# B&R Automation Studio project OpcUaServer_Reading-SessionDiagnosticsArray
Automation Studio 4.9

## Configuration Config1

CPU PC_any, AutomationRuntime L4.93, Build 4.1.2, Vc V4.73.3

### Task classes (Cpu.sw)
```
Cyclic#1:
  Program <- Program.prg
  UASessDiag <- UASessDiag.prg
Binaries: udbdef, FWRules, TCData, sysconf, Role, User, iomap, ashwd, asfw, arconfig, ashwac
Libraries: AsOpcUac, runtime, standard, astime, asieccon
```

### Hardware
```
PC : PC_any v1.1.1.0 (OrderNumber=PC)
  ConfigurationID = uaserver_Config1
  FileDevice1
  FileDeviceName1 = USER
  FileDevicePath1 = USER_PATH
  ActivateOpcUa = 1
  OpcUaPort = 4841
  OpcUaInformationModels_PV_Version = 1
```

## Configuration Config2

CPU X20CP3585, AutomationRuntime J4.93, Build 4.1.2, Vc V4.73.3

### Task classes (Cpu.sw)
```
Cyclic#1:
  Program <- Program.prg
Cyclic#4:
  UASessDiag <- UASessDiag.prg
Libraries: AsIODiag, runtime
```

### Hardware
```
X20CP3585 : X20CP3585 v1.10.0.0
  Connector IF2:
    ActivateDevice = 1
    Mode = Manual
    InternetAddress = 10.24.153.43
    SubnetMask = 255.255.255.192
    ActivateIna = 0
    ActivateSnmp = 2
  ConfigurationID = uaserver_Config2
  FileDevice1
  FileDeviceName1 = USER
  FileDevicePath1 = USER_PATH
  EthernetDefaultGateway = 10.24.153.1
  ActivateOpcUa = 1
  OpcUaInformationModels_PV_Version = 1
```

## Logical view

Binary libraries used (declarations not repeated): operator, runtime, astime, AsIecCon, AsOpcUac, standard, AsIODiag


### Program Logical/Program (IEC)

#### Variables.var
```iecst
VAR
	i : DINT;
END_VAR
```

#### Main.st
```iecst
PROGRAM _INIT
	i := 0;

END_PROGRAM

PROGRAM _CYCLIC
	i := i + 1;

END_PROGRAM

PROGRAM _EXIT
	(* Insert code here *)

END_PROGRAM
```

### Program Logical/UASessDiag (IEC) - Read OPC UA session diagnostic

#### ReadSessionDiagnosticsArray.st - Cyclic code
```iecst
PROGRAM _INIT
	step := RSD_INIT;

	(* NodeId for Root/Objects/Server/ServerDiagnostics/SessionsDiagnosticsSummary/SessionDiagnosticsArray is i=3707. *)
	ServerDiagnosticNodeID.NamespaceIndex := 0;
	ServerDiagnosticNodeID.IdentifierType := UAIdentifierType_Numeric;
	ServerDiagnosticNodeID.Identifier := '3707';

	ServerDiagnosticVariable := 'SessionDiagnosticsArray';
	SessionDiagnosticsArray;
	tonRepeat.PT := T#5s;

	timeout := T#5s;
END_PROGRAM

PROGRAM _CYCLIC
	CASE step OF
		RSD_INIT:
		ErrorID := 0;
		IF DiagCpuIsSimulated() THEN
			fbUAConnect.ServerEndpointUrl := 'opc.tcp://localhost:4841';
		ELSE
			fbUAConnect.ServerEndpointUrl := 'opc.tcp://localhost:4840';
		END_IF
		fbUAConnect( Execute := FALSE,
				SessionConnectInfo := SessionConnectInfo,
				Timeout := timeout,
		); // reset fb
		fbUAConnect( Execute := TRUE );
		step := RSD_W_CONNECT;

		RSD_W_CONNECT:
		IF fbUAConnect.Done THEN (* ok *)
			fbUaNodeGetHandle( Execute := FALSE,
							ConnectionHdl := fbUAConnect.ConnectionHdl,
							NodeID := ServerDiagnosticNodeID,
							Timeout := timeout );
			fbUaNodeGetHandle( Execute := TRUE );
			fbUAConnect( Execute := FALSE ); (* reset fb *)
			step := RSD_W_NODE_HANDLE;
		ELSIF fbUAConnect.Error THEN (* error *)
			ErrorID := fbUAConnect.ErrorID;
			fbUAConnect( Execute := FALSE ); (* reset fb *)
			step := RSD_ERROR_CONNECT_TO_SERVER;
		ELSE (* busy *)
			fbUAConnect();
		END_IF

		RSD_W_NODE_HANDLE:
		IF fbUaNodeGetHandle.Done THEN (* ok *)
			fbUaRead( ConnectionHdl := fbUAConnect.ConnectionHdl,
					  NodeHdl := fbUaNodeGetHandle.NodeHdl,
					  Variable := ServerDiagnosticVariable,
					  Timeout := timeout
					);
			fbUaRead( Variable := ServerDiagnosticVariable, Execute := TRUE );
			fbUaNodeGetHandle( Execute := FALSE ); (* reset fb *)
			step := RSD_W_DIAGNOSTIC_READ;
		ELSIF fbUaNodeGetHandle.Error THEN (* error *)
			ErrorID := fbUaNodeGetHandle.Error;
			fbUaNodeGetHandle( Execute := FALSE ); (* reset fb *)
			step := RSD_ERROR_GET_NODE_HANDLE;
		ELSE (* busy *)
			fbUaNodeGetHandle();
		END_IF

		RSD_W_DIAGNOSTIC_READ:
		IF fbUaRead.Done THEN (* ok *)
			fbUaRead( Variable := ServerDiagnosticVariable, Execute := FALSE );
			tonRepeat( IN := FALSE );

			step := RSD_W_START_READING;
		ELSIF fbUaRead.Error THEN (* error *)
			ErrorID := fbUaRead.ErrorID;
			fbUaRead( Variable := ServerDiagnosticVariable, Execute := FALSE );
			step := RSD_ERROR_READ_DIAGNOSTIC;
		ELSE (* busy *)
			fbUaRead( Variable := ServerDiagnosticVariable );
		END_IF

		RSD_W_START_READING:
		tonRepeat( IN := TRUE );
		IF tonRepeat.Q THEN
			fbUaRead( Variable := ServerDiagnosticVariable, Execute := TRUE );
			step := RSD_W_DIAGNOSTIC_READ;
		END_IF

		RSD_ERROR_CONNECT_TO_SERVER:
		RSD_ERROR_GET_NODE_HANDLE:
		RSD_ERROR_READ_DIAGNOSTIC:

	END_CASE

END_PROGRAM

PROGRAM _EXIT
END_PROGRAM
```

#### ReadSessionDiagnosticsArray.typ - Local data types
```iecst
TYPE
	RsdaStepType :
		(
		RSD_INIT,
		RSD_W_CONNECT,
		RSD_W_NODE_HANDLE,
		RSD_W_DIAGNOSTIC_READ,
		RSD_W_START_READING,
		RSD_ERROR_CONNECT_TO_SERVER,
		RSD_ERROR_GET_NODE_HANDLE,
		RSD_ERROR_READ_DIAGNOSTIC
		);
	ApplicationTypeEnum :
		(
		ApplicationType_Server,
		ApplicationType_Client,
		ApplicationType_ClientAndServer,
		ApplicationType_DiscoveryServer
		);
	ApplicationDescription : 	STRUCT
		ApplicationUri : STRING[255];
		ProductUri : STRING[255];
		ApplicationName : UALocalizedText;
		ApplicationType : ApplicationTypeEnum;
		GatewayServerUri : STRING[255];
		DiscoveryProfileUri : STRING[255];
		DiscoveryUrlsLength : UANoOfElements;
		DiscoveryUrls : ARRAY[0..9]OF STRING[255];
	END_STRUCT;
	ServiceCounterDataType : 	STRUCT
		TotalCount : UDINT;
		ErrorCount : UDINT;
	END_STRUCT;
	SessionDiagnosticsDataType : 	STRUCT
		SessionId : UANodeID;
		SessionName : STRING[255];
		ClientDescription : ApplicationDescription;
		ServerUri : STRING[255];
		EndpointUrl : STRING[255];
		LocaleIdsCount : UANoOfElements;
		LocaleIds : ARRAY[0..4]OF STRING[7];
		ActualSessionTimeout : LREAL;
		MaxResponseMessageSize : UDINT;
		ClientConnectionTime : DATE_AND_TIME;
		ClientLasstContactTime : DATE_AND_TIME;
		CurrentSubscriptionsCount : UDINT;
		CurrentMonitoredItemsCount : UDINT;
		CurrentPublishRequestsInQueue : UDINT;
		TotalRequestCount : ServiceCounterDataType;
		UnauthorizedRequestCount : UDINT;
		ReadCount : ServiceCounterDataType;
		HistoryReadCount : ServiceCounterDataType;
		WriteCount : ServiceCounterDataType;
		HistoryUpdateCount : ServiceCounterDataType;
		CallCount : ServiceCounterDataType;
		CreateMonitoredItemsCount : ServiceCounterDataType;
		ModifyMonitoredItemsCount : ServiceCounterDataType;
		SetMonitoringModeCount : ServiceCounterDataType;
		SetTriggeringCount : ServiceCounterDataType;
		DeleteMonitoredItemsCount : ServiceCounterDataType;
		CreateSubscriptionCount : ServiceCounterDataType;
		ModifySubscriptionCount : ServiceCounterDataType;
		SetPublishingModeCount : ServiceCounterDataType;
		PublishCount : ServiceCounterDataType;
		RepublishCount : ServiceCounterDataType;
		TransferSubscriptionsCount : ServiceCounterDataType;
		DeleteSubscriptionsCount : ServiceCounterDataType;
		AddNodesCount : ServiceCounterDataType;
		AddReferencesCount : ServiceCounterDataType;
		DeleteNodesCount : ServiceCounterDataType;
		DeleteReferencesCount : ServiceCounterDataType;
		BrowseCount : ServiceCounterDataType;
		BrowseNextCount : ServiceCounterDataType;
		TranslateBrowsePathToNodeIdCount : ServiceCounterDataType;
		QueryFirstCount : ServiceCounterDataType;
		QueryNextCount : ServiceCounterDataType;
		RegisterNodesCount : ServiceCounterDataType;
		UnregisterNodesCount : ServiceCounterDataType;
	END_STRUCT;
	SessionDiagnosticsArrayType : 	STRUCT
		Length : UAArrayLength;
		Data : ARRAY[0..9]OF SessionDiagnosticsDataType;
	END_STRUCT;
END_TYPE
```

#### ReadSessionDiagnosticsArray.var - Local variables
```iecst
VAR
	fbUAConnect : UA_Connect;
	SessionDiagnosticsArrayHdl : DWORD;
	SessionDiagnosticsArray : SessionDiagnosticsArrayType;
	fbUaNodeGetHandle : UA_NodeGetHandle;
	fbUaRead : UA_Read;
	step : RsdaStepType;
	SessionConnectInfo : UASessionConnectInfo;
	ErrorID : DWORD;
	ServerDiagnosticNodeID : UANodeID;
	timeout : TIME;
	ServerDiagnosticVariable : STRING[255];
	tonRepeat : TON;
END_VAR
```

Listed in the project but not available here: Logical/Global.typ, Logical/Global.var
